FUNCTION_BLOCK FB_MultiZPWM
VAR_INPUT
END_VAR
VAR_OUTPUT
END_VAR
VAR
	bSafety AT %I* 	: BOOL;
	aEnable AT %Q* 	: ARRAY[1..2] OF USINT;
	aValue AT %Q* 	: ARRAY[1..2] OF UINT;
	aCycle			: ARRAY[1..3] OF USINT;
	i				: USINT;	
END_VAR

//Wenn spätestens nach 2 Zyklen kein Ein mehr kommmt, dann ausschalten
FOR i:= 1 TO 3 BY 1 DO
	aCycle[i] := SHR(aCycle[i],1);
	IF aCycle[i].0 AND bSafety THEN
		aEnable[i] := 1;
	ELSE
		aEnable[i] := 0;
	END_IF
END_FOR

METHOD FB_init : BOOL
VAR_INPUT
	bInitRetains : BOOL; // if TRUE, the retain variables are initialized (warm start / cold start)
	bInCopyCode : BOOL;  // if TRUE, the instance afterwards gets moved into the copy code (online change)
END_VAR
IF NOT (F_GetMappingStatus(ADR(bSafety),SIZEOF(bSafety)) = EPlcMappingStatus.MS_Partial) THEN
	bSafety := TRUE;
END_IF
END_METHOD

METHOD M_GetState : BOOL
VAR_INPUT
	nChannel : USINT;
END_VAR
IF nChannel >= 1 AND nChannel <= 2 THEN
	M_GetState := USINT_TO_BOOL(aEnable[nChannel]);
END_IF
END_METHOD

METHOD M_Off
VAR_INPUT
	nChannel : USINT;
END_VAR
IF nChannel >= 1 AND nChannel <= 2 THEN
	aCycle[nChannel] := 0;
	aEnable[nChannel] := 0;
	aValue[nChannel] := 0;
END_IF
END_METHOD

METHOD M_On
VAR_INPUT
	nChannel : USINT;
	nValue	 : UINT;	//Tastverhältnis in 1/10tel % 
END_VAR
//Wenn spätestens nach 2 Zyklen kein Ein mehr kommmt, dann ausschalten
IF nChannel >= 1 AND nChannel <= 2 THEN
	aCycle[nChannel] := 3;
	aValue[nChannel] := REAL_TO_UINT(1023.0 / 100.0 * (UINT_TO_REAL(nValue)/10.0));
END_IF
END_METHOD

END_FUNCTION_BLOCK

(* stored: Version 1.1.0.1, ProductVersion 3.1.4024.6
   POU FB_MultiZPWM: Id {d0e2783e-0dc5-45ca-b945-84241d3fc9b6}, SpecialFunc None
   Method FB_init: Id {64605a5f-7cfc-4516-90c4-92cb5db30cfd}
   Method M_GetState: Id {46412333-7437-4aae-8fa8-a04894c567a7}
   Method M_Off: Id {1dada1a0-788c-4555-9387-74ed55bdd6f2}
   Method M_On: Id {a18ec223-15ba-4109-8dad-f57e1521502f} *)
